// TIA Portal V20 export
DATA_BLOCK "MP108"   // DB310
// stored: MemoryReserve 100
   VAR
      "10 TON SERVO PRESS-1 Z-AXIS EMS&STO SIGNAL" : Bool;
      "10 TON SERVO PRESS-1 Z-AXIS - PROBE 1" : Bool;
      "10 TON SERVO PRESS-2 Z-AXIS EMS&STO SIGNAL" : Bool;
      "10 TON SERVO PRESS-2 Z-AXIS - PROBE 1" : Bool;
      "3 TON SERVO PRESS Z-AXIS EMS&STO SIGNAL" : Bool;
      "3 TON SERVO PRESS Z-AXIS - PROBE 1" : Bool;
      SPARE : Bool;
      SPARE_1 : Bool;
   END_VAR
BEGIN
END_DATA_BLOCK
